Omron Sysmac Studio project progetto_roma_Recuperato (Sysmac Studio 1.56.0.11, StandardProject)

# Controller new_Controller_0: NX1P2-9024DT1 version 1.64
Task PrimaryTask (priority 4, period or condition 2000): Programma0

VAR_GLOBAL
    FL1 : BOOL := False;  (* at BuiltInIO://cpu/#0/Input_Bit_00 *)
    avanti : BOOL := False;  (* at BuiltInIO://cpu/#0/Output_Bit_00 *)
    arrivato_al_gusto : BOOL;
    pompa_bicchiere_avanti : BOOL;
    pompa_bicchiere_indietro : BOOL;
    FL2 : BOOL;
    quantita_necessaria_erogata : BOOL := True;
    FC2 : BOOL;
    lamp_fine : BOOL;
    btn_bevanda_scelta : BOOL;
END_VAR

PROGRAM Programma0
VAR
    stato : INT := 0;
    Timer_bicchiere : TON;
    trigger_timer : BOOL;
    tempo_trascorso_timer_bicchiere : TIME;
    timer_bicchiere_finito : BOOL;
    timer_bicchiere_set : TIME;
END_VAR
VAR_EXTERNAL
    FL1 : BOOL;
    avanti : BOOL;
    arrivato_al_gusto : BOOL;
    pompa_bicchiere_avanti : BOOL;
    pompa_bicchiere_indietro : BOOL;
    FL2 : BOOL;
    quantita_necessaria_erogata : BOOL;
    FC2 : BOOL;
    lamp_fine : BOOL;
    btn_bevanda_scelta : BOOL;
END_VAR
CASE stato OF 
	
	0: //scelta bevanda stop
	avanti := FALSE;
	IF btn_bevanda_scelta THEN
		stato := 1;
	END_IF;
	
	1: //avanti
	avanti := TRUE;
	IF arrivato_al_gusto THEN
		stato := 2;
	ELSIF FC2 THEN
		lamp_fine := TRUE; 
		stato := 0;
	END_IF;
	
	2://pompa su
	avanti := FALSE;
	timer_bicchiere_set := T#1s;
	trigger_timer := TRUE;
	pompa_bicchiere_avanti := TRUE;
	pompa_bicchiere_indietro := FALSE;
	IF timer_bicchiere_finito THEN
		trigger_timer := FALSE;
		stato := 4;
	END_IF;

	4: //bicchiere fermo erogazione liquido
	avanti := FALSE;
	timer_bicchiere_set := T#1s;
	trigger_timer := TRUE;
	pompa_bicchiere_avanti := FALSE;
	pompa_bicchiere_indietro := FALSE;
	IF timer_bicchiere_finito THEN
		trigger_timer := FALSE;
		stato := 3;
	END_IF;
	
	3://pompa_giu
	avanti := FALSE;
	timer_bicchiere_set := T#1s;
	trigger_timer := TRUE;
	pompa_bicchiere_avanti := FALSE;
	pompa_bicchiere_indietro := TRUE;
	IF timer_bicchiere_finito THEN
		trigger_timer := FALSE;
		stato := 5;
	END_IF;
	
	5: 
	avanti := FALSE;
	pompa_bicchiere_avanti := FALSE;
	pompa_bicchiere_indietro := FALSE;
	IF quantita_necessaria_erogata THEN
		stato := 1;
		arrivato_al_gusto := FALSE;
	ELSIF NOT quantita_necessaria_erogata THEN
		trigger_timer := TRUE;
		timer_bicchiere_set := T#2s;
	END_IF;
	
	IF timer_bicchiere_finito THEN
		trigger_timer := FALSE;
		stato := 2;
	END_IF;
	
END_CASE;

Timer_bicchiere(In:=trigger_timer, PT:=timer_bicchiere_set, Q=>timer_bicchiere_finito, ET=>tempo_trascorso_timer_bicchiere);
END_PROGRAM

# Device HMI_NA5_0 (NA): not converted